% RSLogix 500 project WATER_TANK2.RSS, saved by version 8.30.00.16 %
PROJECT "WATER_TA"    % processor: Bul.1763 MicroLogix 1100 Series B %

PROGRAM FILES
  LAD 2   13 rungs

DATA FILES
  O0 OUTPUT  4 elements
  I1 INPUT  6 elements
  S2 STATUS  66 elements
  B3 BINARY  1 elements
  T4 TIMER  2 elements
  C5 COUNTER  1 elements
  R6 CONTROL  1 elements
  N7 INTEGER  1 elements
  F8 FLOAT  1 elements

LADDER 2
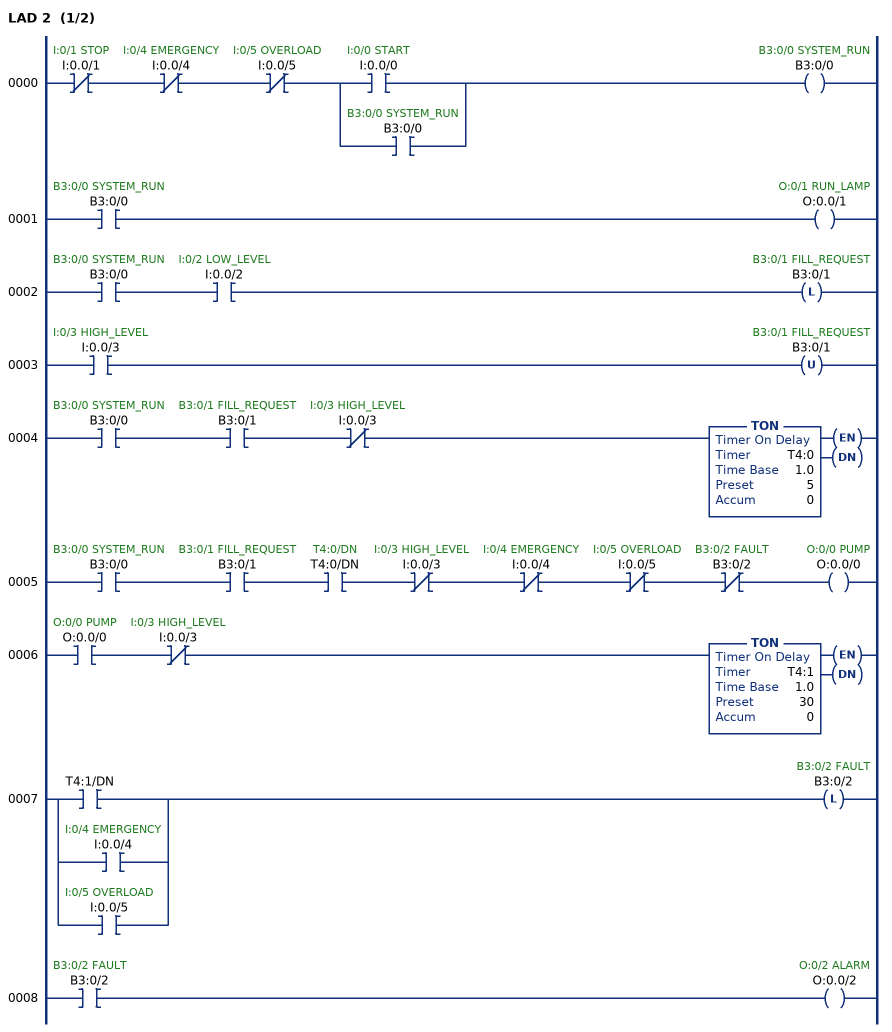
% Rung: 0 %
SOR XIO I:0.0/1 XIO I:0.0/4 XIO I:0.0/5 BST XIC I:0.0/0 NXB XIC B3:0/0 BND OTE B3:0/0 EOR
%   I:0.0/1  STOP  "I:0/1" %
%   I:0.0/4  EMERGENCY  "I:0/4" %
%   I:0.0/5  OVERLOAD  "I:0/5" %
%   I:0.0/0  START  "I:0/0" %
%   B3:0/0  SYSTEM_RUN  "B3:0/0" %
% Rung: 1 %
SOR XIC B3:0/0 OTE O:0.0/1 EOR
%   B3:0/0  SYSTEM_RUN  "B3:0/0" %
%   O:0.0/1  RUN_LAMP  "O:0/1" %
% Rung: 2 %
SOR XIC B3:0/0 XIC I:0.0/2 OTL B3:0/1 EOR
%   B3:0/0  SYSTEM_RUN  "B3:0/0" %
%   I:0.0/2  LOW_LEVEL  "I:0/2" %
%   B3:0/1  FILL_REQUEST  "B3:0/1" %
% Rung: 3 %
SOR XIC I:0.0/3 OTU B3:0/1 EOR
%   I:0.0/3  HIGH_LEVEL  "I:0/3" %
%   B3:0/1  FILL_REQUEST  "B3:0/1" %
% Rung: 4 %
SOR XIC B3:0/0 XIC B3:0/1 XIO I:0.0/3 TON T4:0 1.0 5 0 EOR
%   B3:0/0  SYSTEM_RUN  "B3:0/0" %
%   B3:0/1  FILL_REQUEST  "B3:0/1" %
%   I:0.0/3  HIGH_LEVEL  "I:0/3" %
% Rung: 5 %
SOR XIC B3:0/0 XIC B3:0/1 XIC T4:0/DN XIO I:0.0/3 XIO I:0.0/4 XIO I:0.0/5 XIO B3:0/2 OTE O:0.0/0 EOR
%   B3:0/0  SYSTEM_RUN  "B3:0/0" %
%   B3:0/1  FILL_REQUEST  "B3:0/1" %
%   T4:0/DN  "T4:0/DN" %
%   I:0.0/3  HIGH_LEVEL  "I:0/3" %
%   I:0.0/4  EMERGENCY  "I:0/4" %
%   I:0.0/5  OVERLOAD  "I:0/5" %
%   B3:0/2  FAULT  "B3:0/2" %
%   O:0.0/0  PUMP  "O:0/0" %
% Rung: 6 %
SOR XIC O:0.0/0 XIO I:0.0/3 TON T4:1 1.0 30 0 EOR
%   O:0.0/0  PUMP  "O:0/0" %
%   I:0.0/3  HIGH_LEVEL  "I:0/3" %
% Rung: 7 %
SOR BST BST XIC T4:1/DN NXB XIC I:0.0/4 BND NXB XIC I:0.0/5 BND OTL B3:0/2 EOR
%   I:0.0/4  EMERGENCY  "I:0/4" %
%   I:0.0/5  OVERLOAD  "I:0/5" %
%   B3:0/2  FAULT  "B3:0/2" %
% Rung: 8 %
SOR XIC B3:0/2 OTE O:0.0/2 EOR
%   B3:0/2  FAULT  "B3:0/2" %
%   O:0.0/2  ALARM  "O:0/2" %

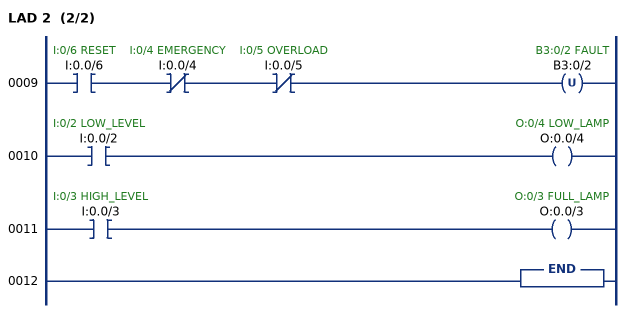
% Rung: 9 %
SOR XIC I:0.0/6 XIO I:0.0/4 XIO I:0.0/5 OTU B3:0/2 EOR
%   I:0.0/6  RESET  "I:0/6" %
%   I:0.0/4  EMERGENCY  "I:0/4" %
%   I:0.0/5  OVERLOAD  "I:0/5" %
%   B3:0/2  FAULT  "B3:0/2" %
% Rung: 10 %
SOR XIC I:0.0/2 OTE O:0.0/4 EOR
%   I:0.0/2  LOW_LEVEL  "I:0/2" %
%   O:0.0/4  LOW_LAMP  "O:0/4" %
% Rung: 11 %
SOR XIC I:0.0/3 OTE O:0.0/3 EOR
%   I:0.0/3  HIGH_LEVEL  "I:0/3" %
%   O:0.0/3  FULL_LAMP  "O:0/3" %
% Rung: 12 %
SOR END EOR

OTHER DOCUMENTED ADDRESSES
  A  "O:0/1"
  D  "I:0/5"
  L  "I:0/5"
  O  "I:0/0"
  Q0:0  "O:0/1"
  S  "B3:0/0"

REVISION NOTES
  0: Last

DATA TABLE (non-zero values as saved)
DATA T4
% .PRE .ACC %
% T4:0 % 5 0
% T4:1 % 30 0
